% RSLogix 500 project START_STOP_LATCH_MOTOR.RSS, saved by version 8.30.00.16 %
PROJECT "UNTITLED"    % processor: Bul.1763 MicroLogix 1100 Series B %

PROGRAM FILES
  LAD 2   3 rungs

DATA FILES
  O0 OUTPUT  4 elements
  I1 INPUT  6 elements
  S2 STATUS  66 elements
  B3 BINARY  1 elements
  T4 TIMER  1 elements
  C5 COUNTER  1 elements
  R6 CONTROL  1 elements
  N7 INTEGER  1 elements
  F8 FLOAT  1 elements

LADDER 2
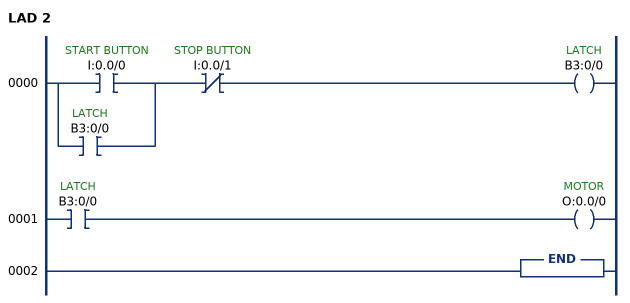
% Rung: 0 %
SOR BST XIC I:0.0/0 NXB XIC B3:0/0 BND XIO I:0.0/1 OTE B3:0/0 EOR
%   I:0.0/0  "START BUTTON" %
%   B3:0/0  "LATCH" %
%   I:0.0/1  "STOP BUTTON" %
% Rung: 1 %
SOR XIC B3:0/0 OTE O:0.0/0 EOR
%   B3:0/0  "LATCH" %
%   O:0.0/0  "MOTOR" %
% Rung: 2 %
SOR END EOR

OTHER DOCUMENTED ADDRESSES
  I:1.0/0  "START BUTTON"

REVISION NOTES
  0: Moved stop button to outside of branch
